RoboDK station: UR5_station_default.rdk

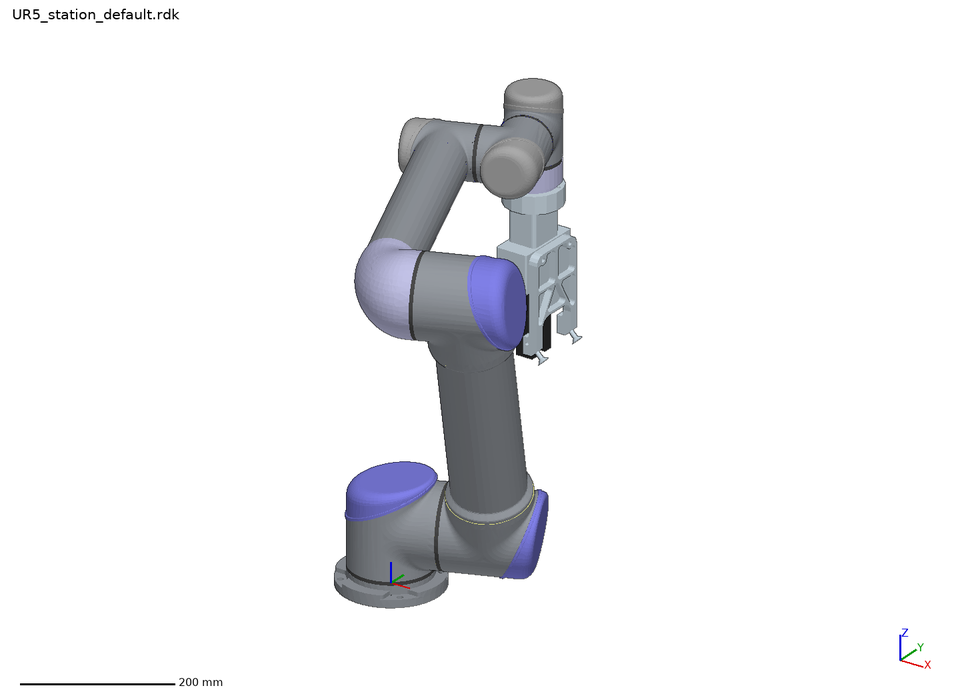
[picture v0: the station drawn from its stored meshes, robots at their saved joint values, targets as dots, program paths as lines]
Station UR5_station_default (saved by RoboDK 5.2.1). Poses are relative to the parent item; angles as X-Y-Z fixed-axis rotations.
Station parameters (name, value as stored): Gripper, 0, CollisionFreePlanner, UR5, CollisionFreePlanner-Rob UR5
  - frame UR5 Base at (0, 0, 0) mm
    - robot UR5: 6 axes, payload 5 kg, reach 850 mm, repeatability 0.1 mm, weight 18.4 kg
        modified DH rows (alpha deg, a mm, theta deg, d mm): 0, 0, 0, 89.2; 90, 0, 180, 0; 0, 425, 0, 0; 0, 392.43, 0, 109; -90, 0, 0, 93.65; 90, 0, 180, 82
        joint limits [-360, -180, -180, -360, -360, -360] to [360, 0, 180, 0, 360, 360]; home [0, -90, -90, 0, 90, 0]; saved at [111.894, -70.08, -107.55, -92.37, 90, 291.894]
      - tool Gripper, TCP at (0, 0, 240) mm, rotated rx 0 ry 0 rz -90 deg, size 100 x 89.2 x 240.5 mm
    - frame FrameN at (0, 0, 0) mm
    - object Table at (-250, 600, 0) mm, rotated rx 0 ry 0 rz -180 deg, size 600 x 1350 x 100 mm, geometry from RhinoPart.ply
